FUNCTION F_ResetErrorList 
VAR_INPUT
	FirstElement : POINTER TO ST_Error;
	NumElements : UDINT;
END_VAR
VAR
	i : UDINT;
	Instance : POINTER TO ST_Error;
END_VAR

IF FirstElement = 0 THEN 
	RETURN;
END_IF


FOR i := 0 TO (NUMElements - 1) BY 1 DO
	Instance := FirstElement + (i*SIZEOF(firstelement^));
	Instance^.Active := FALSE;
END_FOR

END_FUNCTION

(* stored: Version 1.1.0.1, ProductVersion 3.1.4024.12
   POU F_ResetErrorList: Id {ceef1906-f954-4e02-b511-088951be0730}, SpecialFunc None *)
